// Core §3.8a/§3.10.2 — persistent configuration ownership class.
// Ordinals are an append-only PLC/HMI transport contract.
{attribute 'qualified_only'}
TYPE E_ConfigKind :
(
    PAR_CFG     := 0,
    STATION_CFG := 1,
    LINE_CFG    := 2      // §3.8e shared by every station on a line; one owner
) DINT;
END_TYPE

(* stored: Version 1.1.0.1, ProductVersion 3.1.4024.12
   DUT E_ConfigKind: Id {2d2baf35-931d-4fb0-9704-7afad63e8448} *)
